FUNCTION_BLOCK ABSTRACT FB_MotionAxisStageAbstract IMPLEMENTS I_MotionAxisStage
VAR
END_VAR

END_FUNCTION_BLOCK

(* stored: Version 1.1.0.1
   POU FB_MotionAxisStageAbstract: Id {44e1c05d-0254-4ddf-bbd0-905230ca599d}, SpecialFunc None *)
